Universal Robots PolyScope program: Pour_spoon.urp

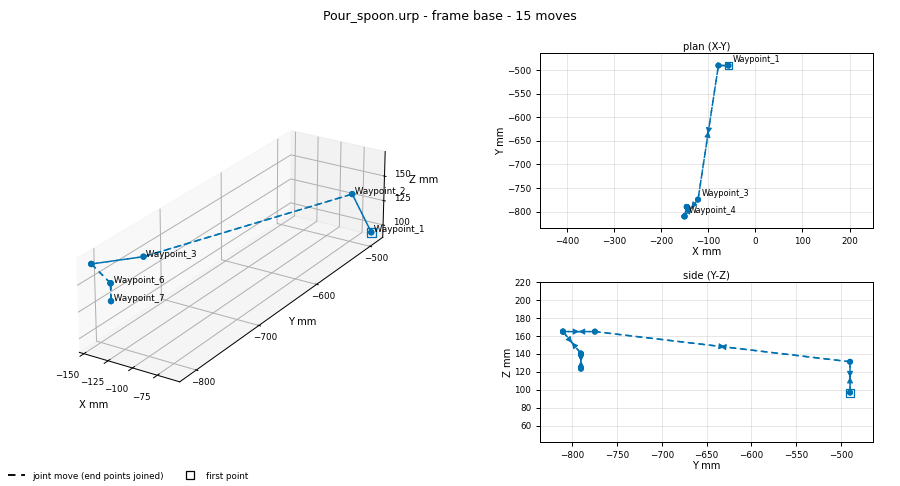
[picture p0: tool path of Pour_spoon.urp in frame base, 15 of 15 moves have a stored position in this frame; points joined in program order, loops and branches not executed]
Program Pour_spoon (installation=default directory=/programs/Matcha createdIn=5.12.6.1102099 lastSavedIn=5.12.6.1102099 robotSerialNumber=20215500597)
Calibrated DH parameters: a=[0.000193, -0.066673, -0.391568, -0.000012, 0.00005, 0]; d=[0.162643, -472.05677, 465.132521, 7.058239, 0.099746, 0.099582]; alpha=[1.571116, 0.00089, 0.003862, 1.569269, -1.569248, 0]; deltaTheta=[0, -1.413394, 7.628392, 0.068187, 0, -0.000001]
Robot Program (runOnlyOnce=true)
  MoveJ speed 60 deg/s, acceleration 80 deg/s^2 (useActiveTCP=true) feature=Base
    Waypoint Waypoint_1: TCP in base x=-57.013 y=-490.112 z=96.992 mm, rx=-0.0141 ry=1.5918 rz=-0.0244 rad; joints [41.641, -46.22, 88.995, -44.212, -47.878, -90.494] deg; TCP offset x=0 y=0 z=191.5 mm, rx=0 ry=0 rz=0 rad
    Waypoint Waypoint_2: TCP in base x=-78.434 y=-490.1 z=131.326 mm, rx=0.4805 ry=1.5418 rz=-0.5073 rad; joints [28.066, -64.654, 116.746, -54.569, -25.798, -89.184] deg
    Waypoint Waypoint_3: TCP in base x=-121.702 y=-774.525 z=164.941 mm, rx=0.5114 ry=1.5349 rz=-0.5372 rad; joints [48.333, -44.036, 73.202, -45.893, -3.514, -74.704] deg
    Waypoint Waypoint_4: TCP in base x=-150.351 y=-810.109 z=164.98 mm, rx=0.5114 ry=1.5349 rz=-0.5373 rad; joints [48.518, -38.15, 61.985, -41.166, -3.351, -74.103] deg
    Waypoint Waypoint_5: TCP in base x=-150.357 y=-810.116 z=164.962 mm, rx=1.7777 ry=0.0096 rz=1.3613 rad; joints [48.518, -38.148, 61.985, -41.169, -3.35, 68.43] deg
    Waypoint Waypoint_6: TCP in base x=-145.446 y=-790.091 z=140.453 mm, rx=1.6664 ry=-0.6858 rz=1.5724 rad; joints [48.149, -45.19, 80.918, -41.441, 11.561, 87.073] deg
    Waypoint Waypoint_7: TCP in base x=-145.478 y=-790.103 z=123.609 mm, rx=1.6663 ry=-0.6859 rz=1.5723 rad; joints [48.148, -43.815, 81.284, -43.169, 11.568, 87.062] deg
    Waypoint Waypoint_6: TCP in base x=-145.446 y=-790.091 z=140.453 mm, rx=1.6664 ry=-0.6858 rz=1.5724 rad; joints [48.149, -45.19, 80.918, -41.441, 11.561, 87.073] deg
    Waypoint Waypoint_7: TCP in base x=-145.478 y=-790.103 z=123.609 mm, rx=1.6663 ry=-0.6859 rz=1.5723 rad; joints [48.148, -43.815, 81.284, -43.169, 11.568, 87.062] deg
    Waypoint Waypoint_6: TCP in base x=-145.446 y=-790.091 z=140.453 mm, rx=1.6664 ry=-0.6858 rz=1.5724 rad; joints [48.149, -45.19, 80.918, -41.441, 11.561, 87.073] deg
    Waypoint Waypoint_5: TCP in base x=-150.357 y=-810.116 z=164.962 mm, rx=1.7777 ry=0.0096 rz=1.3613 rad; joints [48.518, -38.148, 61.985, -41.169, -3.35, 68.43] deg
    Waypoint Waypoint_4: TCP in base x=-150.351 y=-810.109 z=164.98 mm, rx=0.5114 ry=1.5349 rz=-0.5373 rad; joints [48.518, -38.15, 61.985, -41.166, -3.351, -74.103] deg
    Waypoint Waypoint_3: TCP in base x=-121.702 y=-774.525 z=164.941 mm, rx=0.5114 ry=1.5349 rz=-0.5372 rad; joints [48.333, -44.036, 73.202, -45.893, -3.514, -74.704] deg
    Waypoint Waypoint_2: TCP in base x=-78.434 y=-490.1 z=131.326 mm, rx=0.4805 ry=1.5418 rz=-0.5073 rad; joints [28.066, -64.654, 116.746, -54.569, -25.798, -89.184] deg
    Waypoint Waypoint_1: TCP in base x=-57.013 y=-490.112 z=96.992 mm, rx=-0.0141 ry=1.5918 rz=-0.0244 rad; joints [41.641, -46.22, 88.995, -44.212, -47.878, -90.494] deg
